Staubli VAL3: getItem.pgx

program getItem(string& x_sItem[], num x_nIndex)
begin
  x_sItem=sList[x_nIndex]
end
